# EPICS substitutions: db/Beckhoff_1XXX/ecmcEK1501-0010.substitutions
file "ecmcEcSlave.template"
{
  pattern {}
          {}
}

file "ecmcEK1501-0010-ID.template"
{
  pattern {}
          {}
}
